{attribute 'qualified_only'}
VAR_GLOBAL PERSISTENT
	{attribute 'OPC.UA.DA' := '1'}
	Tags: AdsTagsStena;
END_VAR

(* stored: Version 1.1.0.1, ProductVersion 3.1.4024.6
   GVL ADS_Stena: Id {562f9601-fb3e-460e-9881-e3486615fb95} *)
